TYPE ST_DALI_Lamp :
STRUCT
	bManualCtrl		: BOOL;		// if TRUE scenes do not apply
	bLampFailure	: BOOL;		// if TRUE ballast has a lamp problem
	
	nStatus			: BYTE;		// status of a ballast
	
	nLevel			: BYTE;		// 0-255
	
	eKL6821Module	: E_KL6821Module;	//DALI module to which Lamp is connected
	nAddrShort1		: BYTE;				//first 	DALI gear address
	nAddrShort2		: BYTE;				//second 	DALI gear address 
	
	ref_stCommandBuffer	: REFERENCE TO ST_DALIV2CommandBuffer;	//reference to command buffer
	
	//group addresses which DALI_Lamp belongs to
	arrAddrGroup	: ARRAY [1..4] OF BYTE;
	
	//sensors
	bMotionSensor	AT%I*	: BOOL;	//direct info from sensor, edge means movement occured
	bMotionFlag				: BOOL;	//flag keeping info about motion as TRUE for specified period of time
	
END_STRUCT
END_TYPE

(* stored: Version 1.1.0.1, ProductVersion 3.1.4024.5
   DUT ST_DALI_Lamp: Id {a3d69f40-b25c-4fe0-b579-a34b94ed8fa1} *)
